// TIA Portal V17 export
// export: Created 2025-05-22T06:01:47.612155Z, ExportSetting WithDefaults, DisplayName Totally Integrated Automation Portal, DisplayVersion V17 Update 8, DisplayName TIA Portal Openness, DisplayVersion V17 Update 8, DisplayName TIA Portal Version Control Interface, DisplayVersion V17, DisplayName SINAMICS Startdrive Advanced, DisplayVersion V17 SP2, DisplayName SINAMICS Startdrive G110M, G120, G120C, G120D, G120P, G115D, DisplayVersion V17 SP2, DisplayName SINAMICS Startdrive G130, G150, S120, S150, SINAMICS MV, S210, DisplayVersion V17 SP2, DisplayName STEP 7 Professional, DisplayVersion V17 Update 8, DisplayName SINUMERIK ONE STEP 7 Toolbox, DisplayVersion V17 Update 12, DisplayName SINUMERIK ONE PLC Basic Program Plus, DisplayVersion V17 Update 12, DisplayName SINUMERIK 840D sl STEP 7 Toolbox, DisplayVersion V17 Update 12, DisplayName STEP 7 Safety, DisplayVersion V17 Update 6, DisplayName WinCC Advanced, DisplayVersion V17 Update 8
TYPE "UNIT_2_FIXTURE_POSITIONS"
// stored: IsFailsafeCompliant false
   STRUCT
      IN_LOAD_UNLOAD_STATION_1 : Bool;   // UNIT 2 FIXTURE IN LOAD UNLOAD STATION
      IN_MEASURING_STATION_2 : Bool;   // UNIT 2 FIXTURE IN SPARE STATION
      IN_CLADDING_STATION_3 : Bool;   // UNIT 2 FIXTURE IN CLADDING STATION
      IN_CLEAN_STATION_4 : Bool;   // UNIT 2 FIXTURE IN MEASURING/CLEANING STATION
      NO_DEFINED_POSITION : Bool;   // UNIT 2 FIXTURE IN NO DEFINED POSITION
   END_STRUCT;
END_TYPE
